// TIA Portal V17 export
// export: Created 2025-06-26T06:49:27.8171915Z, ExportSetting WithDefaults, DisplayName Totally Integrated Automation Portal, DisplayVersion V17 Update 8, DisplayName TIA Portal Openness, DisplayVersion V17 Update 8, DisplayName TIA Portal Version Control Interface, DisplayVersion V17, DisplayName STEP 7 Professional, DisplayVersion V17 Update 8, DisplayName STEP 7 Safety, DisplayVersion V17 Update 6, DisplayName WinCC Advanced, DisplayVersion V17 Update 8
TYPE "stProcessValve2"
// stored: IsFailsafeCompliant false
   STRUCT
      bOpenRequest : Bool;   // Auto mode command. 1 = open valve, 0 = do nothing
      bCloseRequest : Bool;   // Auto mode command. 1 = close valve, 0 = do nothing
      bOpenStatus : Bool;   // Feedback from valve. 1 = valve is open, 0 = valve is not open
      bClosedStatus : Bool;   // Feedback from valve. 1 = valve is closed, 0 = valve is not closed
      bNormalState : Bool;   // 1 = Normally Open, 0 = Normally Closed
      bOpenCommand : Bool;   // Output to valve. 1 = drive in oipen direction, 0 = do not drive in open direction
      bCloseCommand : Bool;   // Output to valve. 1 = drive in closed direction, 0 = do not drive in closed direction
      bManualMode : Bool;   // 1 = Manual Mode, 0 = not Manual Mode
      bManualOpenRequest : Bool;   // Manual mode command. 1 = open valve, 0 = do nothing
      bManualCloseRequest : Bool;   // Manual mode command. 1 = close valve, 0 = do nothing
      nState : USInt := 0;   // 0 = unknown, 1 = closed, 2 = opening, 3 = open, 4 = closing, 5 = closing error, 6 = opening error
      tOpeningTimeout : Time := T#5s;   // Time to allow for opening before flagging an error
      tClosingTimeout : Time := T#5s;   // Time to allow for closing before flagging an error
   END_STRUCT;
END_TYPE
